// TIA Portal project "Project4" (V17)

(* hardware
DEVICE "S7-1200 station_1"  S7-1200 Station
   slot 0: "Rack_0"  S7-1200 Rack  Rack  V1.0
   slot 1: "PLC_1"  CPU 1212C DC/DC/DC  6ES7 212-1AE40-0XB0  V4.3
DEVICE "HMI_1"  TP1200 Comfort
   slot 0: "HMI_1"  TP1200 Comfort  6AV2 124-0MC01-0AX0  17.0.0.0
   slot 1: "HMI_RT_1"  TP1200 Comfort  6AV2 124-0MC01-0AX0  17.0.0.0
   slot 5: "HMI_1.IE_CP_1"  PROFINET Interface  17.0.0.0
      slot 1: "PROFINET Interface_1"  PROFINET Interface
         slot 1: "Port_1"  Port
         slot 2: "Port_2"  Port
   slot 7: "HMI_1.MPI/DP_CP_1"  MPI/DP Interface  17.0.0.0
*)

// ===== PLC "PLC_1"  CPU 1212C DC/DC/DC =====

VAR_GLOBAL   // PLC tag table "Default tag table"
   "System_Byte" AT %MB1 : Byte;
   "FirstScan" AT %M1.0 : Bool;
   "DiagStatusUpdate" AT %M1.1 : Bool;
   "AlwaysTRUE" AT %M1.2 : Bool;
   "AlwaysFALSE" AT %M1.3 : Bool;
   "Clock_Byte" AT %MB0 : Byte;
   "Clock_10Hz" AT %M0.0 : Bool;
   "Clock_5Hz" AT %M0.1 : Bool;
   "Clock_2.5Hz" AT %M0.2 : Bool;
   "Clock_2Hz" AT %M0.3 : Bool;
   "Clock_1.25Hz" AT %M0.4 : Bool;
   "Clock_1Hz" AT %M0.5 : Bool;
   "Clock_0.625Hz" AT %M0.6 : Bool;
   "Clock_0.5Hz" AT %M0.7 : Bool;
   "Imp1s" AT %M100.0 : Bool;
   "fp_1s" AT %M100.1 : Bool;
   "fp_100ms" AT %M100.2 : Bool;
   "Imp0.1s" AT %M100.3 : Bool;
   "PO1_calc" AT %IW0 : Int;
   "PO2_calc" AT %IW1 : Int;
   "VO1_calc" AT %IW2 : Int;
   "VO2_calc" AT %IW3 : Int;
   "Tag_1" AT %M500.0 : Bool;
   "Tag_2" AT %M500.1 : Bool;
   "Tag_3" AT %M500.2 : Bool;
END_VAR

TYPE "_tSter"
   STRUCT
      Tryb : Bool;
      SterowanieAuto : Bool;
      SterowanieRęka : Bool;
      ZadanaPrędkośćRęka : Int;
      ZadanaPrędkośćAuto : Int;
      PrędkośćWyjściowa : Int;
      Status : Int;
      Wyjscie : Bool;
      CzasWlaczenia : Int;
      Awaria : Bool;
      Ack : Bool;
      "ON/OFF" : Bool;
   END_STRUCT;
END_TYPE

DATA_BLOCK "SterowanieDANE"   // DB1
{ S7_Optimized_Access := 'TRUE' }
VERSION : 0.1
   VAR
      P01 : "_tSter";
      P02 : "_tSter";
      VO1 : "_tSter";
      VO2 : "_tSter";
   END_VAR
BEGIN
   P01.ZadanaPrędkośćAuto := 100;
   P01.PrędkośćWyjściowa := 0;
   P02.ZadanaPrędkośćAuto := 100;
   VO1.ZadanaPrędkośćAuto := 100;
   VO2.ZadanaPrędkośćAuto := 100;
END_DATA_BLOCK

DATA_BLOCK "DB_Zbiornik"   // DB2
{ S7_Optimized_Access := 'TRUE' }
VERSION : 0.1
   VAR
      Poziom : Real;
      LL : Bool;
      LH : Bool;
      PredkoscNapelniania : Int;
      PredkoscOprozniania : Int;
      LM : Bool;
   END_VAR
BEGIN
END_DATA_BLOCK

DATA_BLOCK "Operacje"   // DB4
{ S7_Optimized_Access := 'TRUE' }
VERSION : 0.1
   VAR
      Napelnianie : Bool;
      Oproznianie : Bool;
   END_VAR
BEGIN
END_DATA_BLOCK

DATA_BLOCK "tims"   // DB5
{ S7_Optimized_Access := 'TRUE' }
VERSION : 0.1
   VAR
      ton1 : IEC_TIMER;
      ton2 : IEC_TIMER;
   END_VAR
BEGIN
END_DATA_BLOCK

DATA_BLOCK "Awarie"   // DB6
{ S7_Optimized_Access := 'TRUE' }
VERSION : 0.1
   VAR
      aw : Word;
   END_VAR
BEGIN
END_DATA_BLOCK

// folder: System blocks/Program resources

DATA_BLOCK "IEC_Timer_0_DB"   // DB3
{ S7_Optimized_Access := 'TRUE' }
AUTHOR : Simatic
FAMILY : IEC
NAME : IEC_TMR
VERSION : 1.0
// stored: InstanceOfName IEC_TIMER
"IEC_TIMER"
BEGIN
END_DATA_BLOCK

// folder: (top level)

FUNCTION "FC_Zbiornik" : Void   // FC1, LAD
{ S7_Optimized_Access := 'TRUE' }
VERSION : 0.1
   VAR_IN_OUT
      IEC_Timer_0_Instance : TP_TIME;
   END_VAR
BEGIN

REGION Network 1
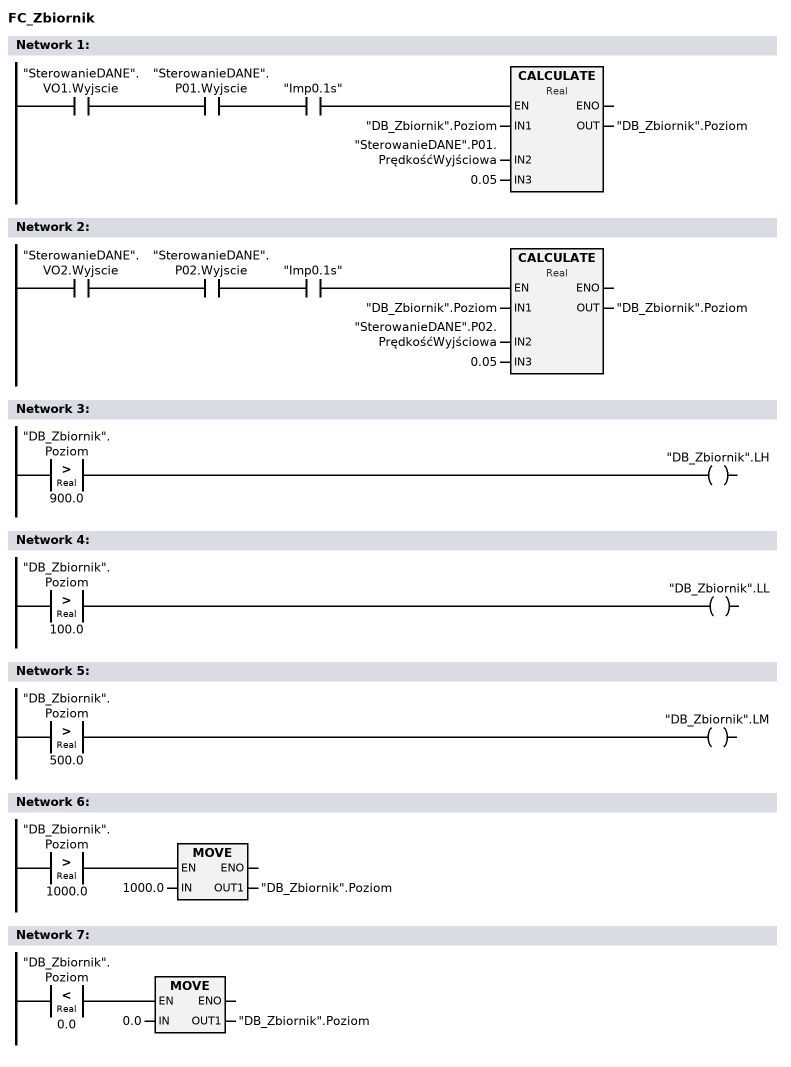
   RUNG wire#powerrail
      Contact( "SterowanieDANE".VO1.Wyjscie )
      Contact( "SterowanieDANE".P01.Wyjscie )
      Contact( "Imp0.1s" )
      { S7_Templates := "SrcType := Real"; S7_Expression := "(IN2 * IN3) + IN1" } Calculate(in1 := "DB_Zbiornik".Poziom, in2 := "SterowanieDANE".P01.PrędkośćWyjściowa, in3 := 0.05, out => "DB_Zbiornik".Poziom)
   END_RUNG
   // the same network as SCL:
   IF "SterowanieDANE".VO1.Wyjscie AND "SterowanieDANE".P01.Wyjscie AND "Imp0.1s" THEN
       "DB_Zbiornik".Poziom := ("SterowanieDANE".P01.PrędkośćWyjściowa * 0.05) + "DB_Zbiornik".Poziom;
   END_IF;
END_REGION

REGION Network 2
   RUNG wire#powerrail
      Contact( "SterowanieDANE".VO2.Wyjscie )
      Contact( "SterowanieDANE".P02.Wyjscie )
      Contact( "Imp0.1s" )
      { S7_Templates := "SrcType := Real"; S7_Expression := "IN1 - (IN2 * IN3)" } Calculate(in1 := "DB_Zbiornik".Poziom, in2 := "SterowanieDANE".P02.PrędkośćWyjściowa, in3 := 0.05, out => "DB_Zbiornik".Poziom)
   END_RUNG
   // the same network as SCL:
   IF "SterowanieDANE".VO2.Wyjscie AND "SterowanieDANE".P02.Wyjscie AND "Imp0.1s" THEN
       "DB_Zbiornik".Poziom := "DB_Zbiornik".Poziom - ("SterowanieDANE".P02.PrędkośćWyjściowa * 0.05);
   END_IF;
END_REGION

REGION Network 3
   RUNG wire#powerrail
      { S7_Templates := "SrcType := Real" } GT_Contact(in1 := "DB_Zbiornik".Poziom, in2 := 900.0)
      Coil( "DB_Zbiornik".LH )
   END_RUNG
   // the same network as SCL:
   "DB_Zbiornik".LH := "DB_Zbiornik".Poziom > 900.0;
END_REGION

REGION Network 4
   RUNG wire#powerrail
      { S7_Templates := "SrcType := Real" } GT_Contact(in1 := "DB_Zbiornik".Poziom, in2 := 100.0)
      Coil( "DB_Zbiornik".LL )
   END_RUNG
   // the same network as SCL:
   "DB_Zbiornik".LL := "DB_Zbiornik".Poziom > 100.0;
END_REGION

REGION Network 5
   RUNG wire#powerrail
      { S7_Templates := "SrcType := Real" } GT_Contact(in1 := "DB_Zbiornik".Poziom, in2 := 500.0)
      Coil( "DB_Zbiornik".LM )
   END_RUNG
   // the same network as SCL:
   "DB_Zbiornik".LM := "DB_Zbiornik".Poziom > 500.0;
END_REGION

REGION Network 6
   RUNG wire#powerrail
      { S7_Templates := "SrcType := Real" } GT_Contact(in1 := "DB_Zbiornik".Poziom, in2 := 1000.0)
      Move(in := 1000.0, out1 => "DB_Zbiornik".Poziom)
   END_RUNG
   // the same network as SCL:
   IF "DB_Zbiornik".Poziom > 1000.0 THEN "DB_Zbiornik".Poziom := 1000.0; END_IF;
END_REGION

REGION Network 7
   RUNG wire#powerrail
      { S7_Templates := "SrcType := Real" } LT_Contact(in1 := "DB_Zbiornik".Poziom, in2 := 0.0)
      Move(in := 0.0, out1 => "DB_Zbiornik".Poziom)
   END_RUNG
   // the same network as SCL:
   IF "DB_Zbiornik".Poziom < 0.0 THEN "DB_Zbiornik".Poziom := 0.0; END_IF;
END_REGION
END_FUNCTION

FUNCTION "Sterowanie" : Void   // FC2, LAD
{ S7_Optimized_Access := 'TRUE' }
VERSION : 0.1
   VAR_INPUT
      ZadanaPrędkośćRęka : Int;
      ZadanaPrędkośćAuto : Int;
      Ack : Bool;
   END_VAR
   VAR_OUTPUT
      PrędkośćWyjściowa : Int;
      Status : Int;
   END_VAR
   VAR_IN_OUT
      "ON/OFF" : Bool;
      Tryb : Bool;
      SterowanieAuto : Bool;
      SterowanieRęka : Bool;
      CzasWlaczenia : Int;
      Awaria : Bool;
      Wyjscie : Bool;
   END_VAR
   VAR_TEMP   // added for the SCL form of the ladder/FBD networks
      _w1 : Bool;
   END_VAR
BEGIN

REGION Network 1: Sterowanie A/R
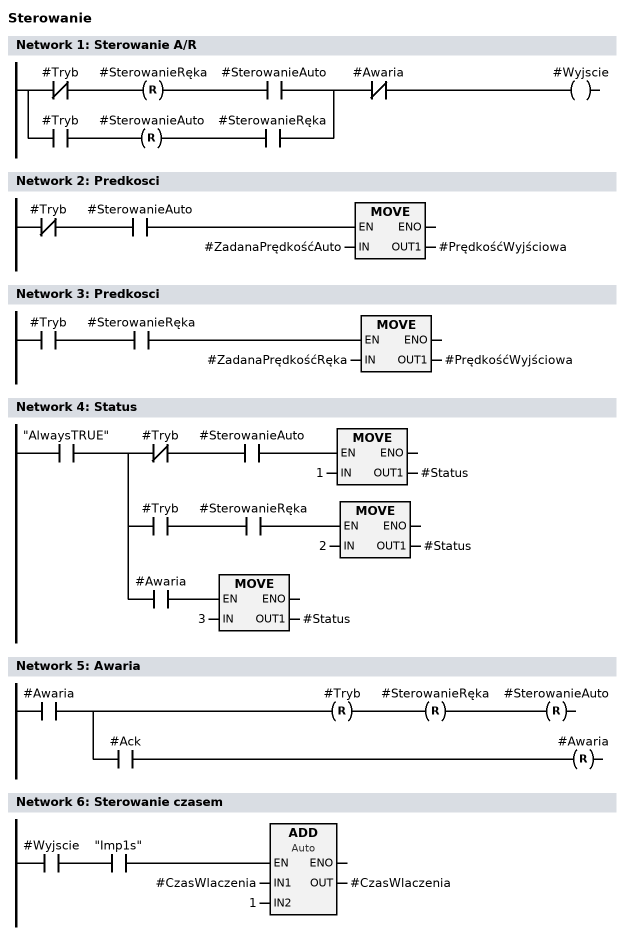
   RUNG wire#powerrail
      I_Contact( #Tryb )
      R_Coil( #SterowanieRęka )
      Contact( #SterowanieAuto )
      wire#w1
      I_Contact( #Awaria )
      Coil( #Wyjscie )
   END_RUNG
   RUNG wire#powerrail
      Contact( #Tryb )
      R_Coil( #SterowanieAuto )
      Contact( #SterowanieRęka )
   END_RUNG wire#w1
   // the same network as SCL:
   IF NOT #Tryb THEN #SterowanieRęka := FALSE; END_IF;
   #_w1 := NOT #Tryb AND #SterowanieAuto;
   IF #Tryb THEN #SterowanieAuto := FALSE; END_IF;
   #Wyjscie := (#_w1 OR (#Tryb AND #SterowanieRęka)) AND NOT #Awaria;
END_REGION

REGION Network 2: Predkosci
   RUNG wire#powerrail
      I_Contact( #Tryb )
      Contact( #SterowanieAuto )
      Move(in := #ZadanaPrędkośćAuto, out1 => #PrędkośćWyjściowa)
   END_RUNG
   // the same network as SCL:
   IF NOT #Tryb AND #SterowanieAuto THEN #PrędkośćWyjściowa := #ZadanaPrędkośćAuto; END_IF;
END_REGION

REGION Network 3: Predkosci
   RUNG wire#powerrail
      Contact( #Tryb )
      Contact( #SterowanieRęka )
      Move(in := #ZadanaPrędkośćRęka, out1 => #PrędkośćWyjściowa)
   END_RUNG
   // the same network as SCL:
   IF #Tryb AND #SterowanieRęka THEN #PrędkośćWyjściowa := #ZadanaPrędkośćRęka; END_IF;
END_REGION

REGION Network 4: Status
   RUNG wire#powerrail
      Contact( "AlwaysTRUE" )
      wire#w1
      I_Contact( #Tryb )
      Contact( #SterowanieAuto )
      Move(in := 1, out1 => #Status)
   END_RUNG
   RUNG wire#w1
      Contact( #Tryb )
      Contact( #SterowanieRęka )
      Move(in := 2, out1 => #Status)
   END_RUNG
   RUNG wire#w1
      Contact( #Awaria )
      Move(in := 3, out1 => #Status)
   END_RUNG
   // the same network as SCL:
   IF "AlwaysTRUE" AND NOT #Tryb AND #SterowanieAuto THEN #Status := 1; END_IF;
   IF "AlwaysTRUE" AND #Tryb AND #SterowanieRęka THEN #Status := 2; END_IF;
   IF "AlwaysTRUE" AND #Awaria THEN #Status := 3; END_IF;
END_REGION

REGION Network 5: Awaria
   RUNG wire#powerrail
      Contact( #Awaria )
      wire#w1
      R_Coil( #Tryb )
      R_Coil( #SterowanieRęka )
      R_Coil( #SterowanieAuto )
   END_RUNG
   RUNG wire#w1
      Contact( #Ack )
      R_Coil( #Awaria )
   END_RUNG
   // the same network as SCL:
   IF #Awaria THEN
       #Tryb := FALSE;
       #SterowanieRęka := FALSE;
       #SterowanieAuto := FALSE;
   END_IF;
   IF #Awaria AND #Ack THEN #Awaria := FALSE; END_IF;
END_REGION

REGION Network 6: Sterowanie czasem
   RUNG wire#powerrail
      Contact( #Wyjscie )
      Contact( "Imp1s" )
      Add(in1 := #CzasWlaczenia, in2 := 1, out => #CzasWlaczenia)
   END_RUNG
   // the same network as SCL:
   IF #Wyjscie AND "Imp1s" THEN #CzasWlaczenia := #CzasWlaczenia + 1; END_IF;
END_REGION
END_FUNCTION

FUNCTION "Napelnianie" : Void   // FC3, LAD
{ S7_Optimized_Access := 'TRUE' }
VERSION : 0.1
BEGIN

REGION Network 1
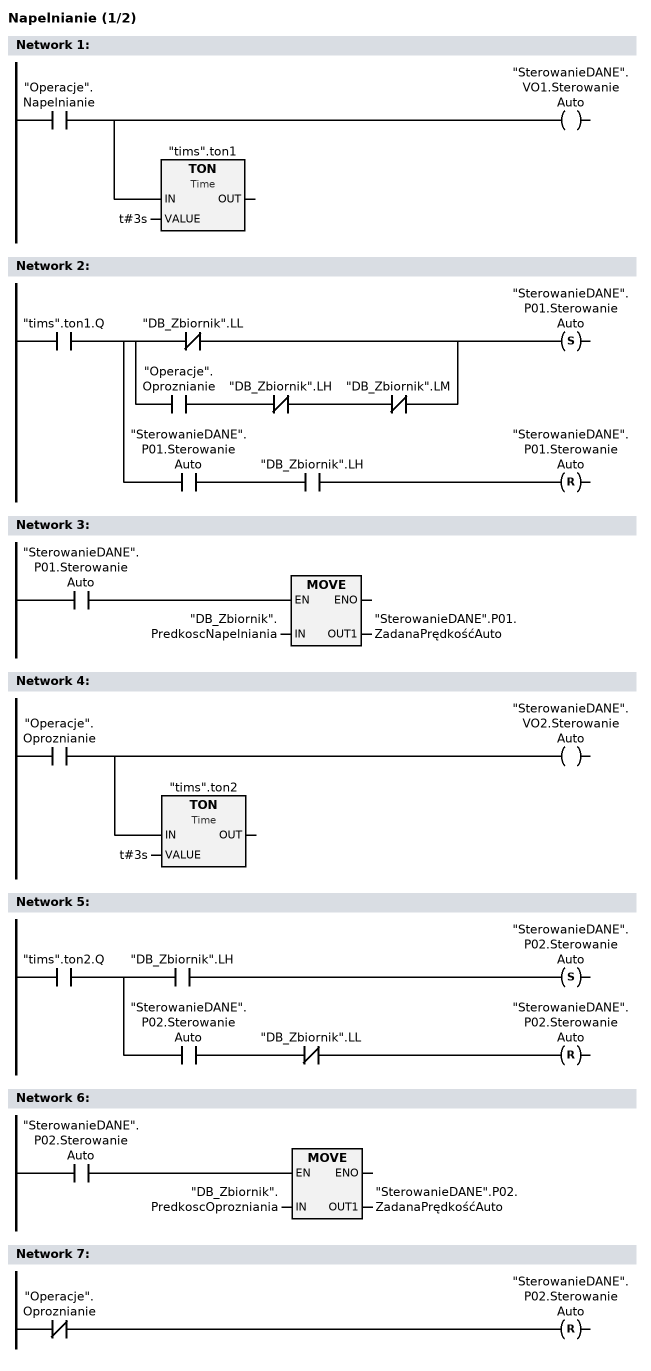
   "SterowanieDANE".VO1.SterowanieAuto := "Operacje".Napelnianie;
   "tims".ton1.TON(IN := "Operacje".Napelnianie, PT := t#3s);   // TON coil
END_REGION

REGION Network 2
   RUNG wire#powerrail
      Contact( "tims".ton1.Q )
      wire#w1
      I_Contact( "DB_Zbiornik".LL )
      wire#w2
      S_Coil( "SterowanieDANE".P01.SterowanieAuto )
   END_RUNG
   RUNG wire#w1
      Contact( "Operacje".Oproznianie )
      I_Contact( "DB_Zbiornik".LH )
      I_Contact( "DB_Zbiornik".LM )
   END_RUNG wire#w2
   RUNG wire#w1
      Contact( "SterowanieDANE".P01.SterowanieAuto )
      Contact( "DB_Zbiornik".LH )
      R_Coil( "SterowanieDANE".P01.SterowanieAuto )
   END_RUNG
   // the same network as SCL:
   IF "tims".ton1.Q AND (NOT "DB_Zbiornik".LL OR ("Operacje".Oproznianie AND NOT "DB_Zbiornik".LH AND NOT "DB_Zbiornik".LM)) THEN
       "SterowanieDANE".P01.SterowanieAuto := TRUE;
   END_IF;
   IF "tims".ton1.Q AND "SterowanieDANE".P01.SterowanieAuto AND "DB_Zbiornik".LH THEN
       "SterowanieDANE".P01.SterowanieAuto := FALSE;
   END_IF;
END_REGION

REGION Network 3
   RUNG wire#powerrail
      Contact( "SterowanieDANE".P01.SterowanieAuto )
      Move(in := "DB_Zbiornik".PredkoscNapelniania, out1 => "SterowanieDANE".P01.ZadanaPrędkośćAuto)
   END_RUNG
   // the same network as SCL:
   IF "SterowanieDANE".P01.SterowanieAuto THEN
       "SterowanieDANE".P01.ZadanaPrędkośćAuto := "DB_Zbiornik".PredkoscNapelniania;
   END_IF;
END_REGION

REGION Network 4
   "SterowanieDANE".VO2.SterowanieAuto := "Operacje".Oproznianie;
   "tims".ton2.TON(IN := "Operacje".Oproznianie, PT := t#3s);   // TON coil
END_REGION

REGION Network 5
   RUNG wire#powerrail
      Contact( "tims".ton2.Q )
      wire#w1
      Contact( "DB_Zbiornik".LH )
      S_Coil( "SterowanieDANE".P02.SterowanieAuto )
   END_RUNG
   RUNG wire#w1
      Contact( "SterowanieDANE".P02.SterowanieAuto )
      I_Contact( "DB_Zbiornik".LL )
      R_Coil( "SterowanieDANE".P02.SterowanieAuto )
   END_RUNG
   // the same network as SCL:
   IF "tims".ton2.Q AND "DB_Zbiornik".LH THEN "SterowanieDANE".P02.SterowanieAuto := TRUE; END_IF;
   IF "tims".ton2.Q AND "SterowanieDANE".P02.SterowanieAuto AND NOT "DB_Zbiornik".LL THEN
       "SterowanieDANE".P02.SterowanieAuto := FALSE;
   END_IF;
END_REGION

REGION Network 6
   RUNG wire#powerrail
      Contact( "SterowanieDANE".P02.SterowanieAuto )
      Move(in := "DB_Zbiornik".PredkoscOprozniania, out1 => "SterowanieDANE".P02.ZadanaPrędkośćAuto)
   END_RUNG
   // the same network as SCL:
   IF "SterowanieDANE".P02.SterowanieAuto THEN
       "SterowanieDANE".P02.ZadanaPrędkośćAuto := "DB_Zbiornik".PredkoscOprozniania;
   END_IF;
END_REGION

REGION Network 7
   RUNG wire#powerrail
      I_Contact( "Operacje".Oproznianie )
      R_Coil( "SterowanieDANE".P02.SterowanieAuto )
   END_RUNG
   // the same network as SCL:
   IF NOT "Operacje".Oproznianie THEN "SterowanieDANE".P02.SterowanieAuto := FALSE; END_IF;
END_REGION

REGION Network 8
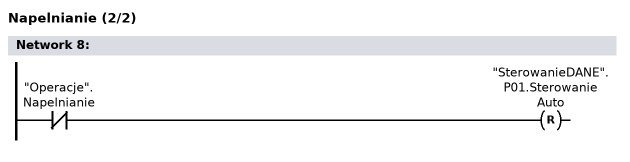
   RUNG wire#powerrail
      I_Contact( "Operacje".Napelnianie )
      R_Coil( "SterowanieDANE".P01.SterowanieAuto )
   END_RUNG
   // the same network as SCL:
   IF NOT "Operacje".Napelnianie THEN "SterowanieDANE".P01.SterowanieAuto := FALSE; END_IF;
END_REGION
END_FUNCTION

ORGANIZATION_BLOCK "Main"   // OB1, LAD, ProgramCycle
TITLE = "Main Program Sweep (Cycle)"
{ S7_Optimized_Access := 'TRUE' }
VERSION : 0.1
   VAR_INPUT
      Initial_Call : Bool;   // Initial call of this OB
      Remanence : Bool;   // =True, if remanent data are available
   END_VAR
   VAR_TEMP   // added for the SCL form of the ladder/FBD networks
      _w1 : Bool;
   END_VAR
BEGIN

REGION Network 1
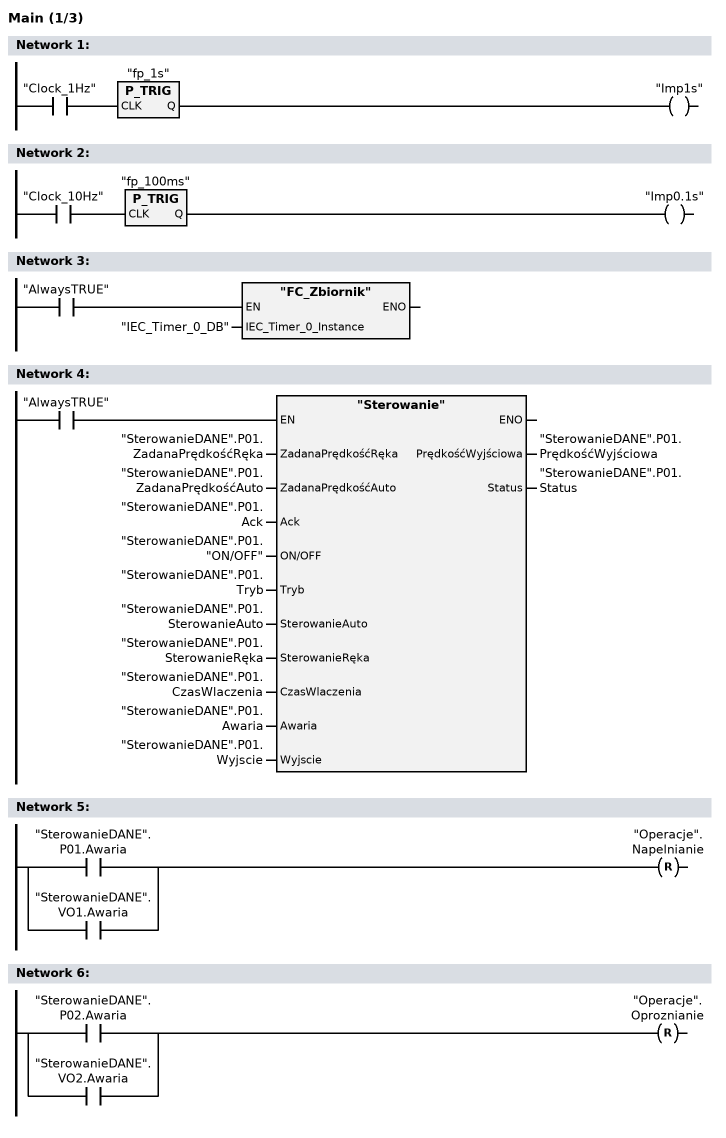
   RUNG wire#powerrail
      Contact( "Clock_1Hz" )
      P_Trig( "fp_1s" )
      Coil( "Imp1s" )
   END_RUNG
   // the same network as SCL:
   #_w1 := "Clock_1Hz" AND NOT "fp_1s";   // rising edge
   "fp_1s" := "Clock_1Hz";
   "Imp1s" := #_w1;
END_REGION

REGION Network 2
   RUNG wire#powerrail
      Contact( "Clock_10Hz" )
      P_Trig( "fp_100ms" )
      Coil( "Imp0.1s" )
   END_RUNG
   // the same network as SCL:
   #_w1 := "Clock_10Hz" AND NOT "fp_100ms";   // rising edge
   "fp_100ms" := "Clock_10Hz";
   "Imp0.1s" := #_w1;
END_REGION

REGION Network 3
   RUNG wire#powerrail
      Contact( "AlwaysTRUE" )
      "FC_Zbiornik"(IEC_Timer_0_Instance := "IEC_Timer_0_DB")
   END_RUNG
   // the same network as SCL:
   IF "AlwaysTRUE" THEN "FC_Zbiornik"(IEC_Timer_0_Instance := "IEC_Timer_0_DB"); END_IF;
END_REGION

REGION Network 4
   RUNG wire#powerrail
      Contact( "AlwaysTRUE" )
      "Sterowanie"(ZadanaPrędkośćRęka := "SterowanieDANE".P01.ZadanaPrędkośćRęka, ZadanaPrędkośćAuto := "SterowanieDANE".P01.ZadanaPrędkośćAuto, Ack := "SterowanieDANE".P01.Ack, "ON/OFF" := "SterowanieDANE".P01."ON/OFF", Tryb := "SterowanieDANE".P01.Tryb, SterowanieAuto := "SterowanieDANE".P01.SterowanieAuto, SterowanieRęka := "SterowanieDANE".P01.SterowanieRęka, CzasWlaczenia := "SterowanieDANE".P01.CzasWlaczenia, Awaria := "SterowanieDANE".P01.Awaria, Wyjscie := "SterowanieDANE".P01.Wyjscie, PrędkośćWyjściowa => "SterowanieDANE".P01.PrędkośćWyjściowa, Status => "SterowanieDANE".P01.Status)
   END_RUNG
   // the same network as SCL:
   IF "AlwaysTRUE" THEN
       "Sterowanie"(ZadanaPrędkośćRęka := "SterowanieDANE".P01.ZadanaPrędkośćRęka,
                    ZadanaPrędkośćAuto := "SterowanieDANE".P01.ZadanaPrędkośćAuto,
                    Ack := "SterowanieDANE".P01.Ack,
                    "ON/OFF" := "SterowanieDANE".P01."ON/OFF",
                    Tryb := "SterowanieDANE".P01.Tryb,
                    SterowanieAuto := "SterowanieDANE".P01.SterowanieAuto,
                    SterowanieRęka := "SterowanieDANE".P01.SterowanieRęka,
                    CzasWlaczenia := "SterowanieDANE".P01.CzasWlaczenia,
                    Awaria := "SterowanieDANE".P01.Awaria,
                    Wyjscie := "SterowanieDANE".P01.Wyjscie,
                    PrędkośćWyjściowa => "SterowanieDANE".P01.PrędkośćWyjściowa,
                    Status => "SterowanieDANE".P01.Status);
   END_IF;
END_REGION

REGION Network 5
   RUNG wire#powerrail
      Contact( "SterowanieDANE".P01.Awaria )
      wire#w1
      R_Coil( "Operacje".Napelnianie )
   END_RUNG
   RUNG wire#powerrail
      Contact( "SterowanieDANE".VO1.Awaria )
   END_RUNG wire#w1
   // the same network as SCL:
   IF "SterowanieDANE".P01.Awaria OR "SterowanieDANE".VO1.Awaria THEN
       "Operacje".Napelnianie := FALSE;
   END_IF;
END_REGION

REGION Network 6
   RUNG wire#powerrail
      Contact( "SterowanieDANE".P02.Awaria )
      wire#w1
      R_Coil( "Operacje".Oproznianie )
   END_RUNG
   RUNG wire#powerrail
      Contact( "SterowanieDANE".VO2.Awaria )
   END_RUNG wire#w1
   // the same network as SCL:
   IF "SterowanieDANE".P02.Awaria OR "SterowanieDANE".VO2.Awaria THEN
       "Operacje".Oproznianie := FALSE;
   END_IF;
END_REGION

REGION Network 7
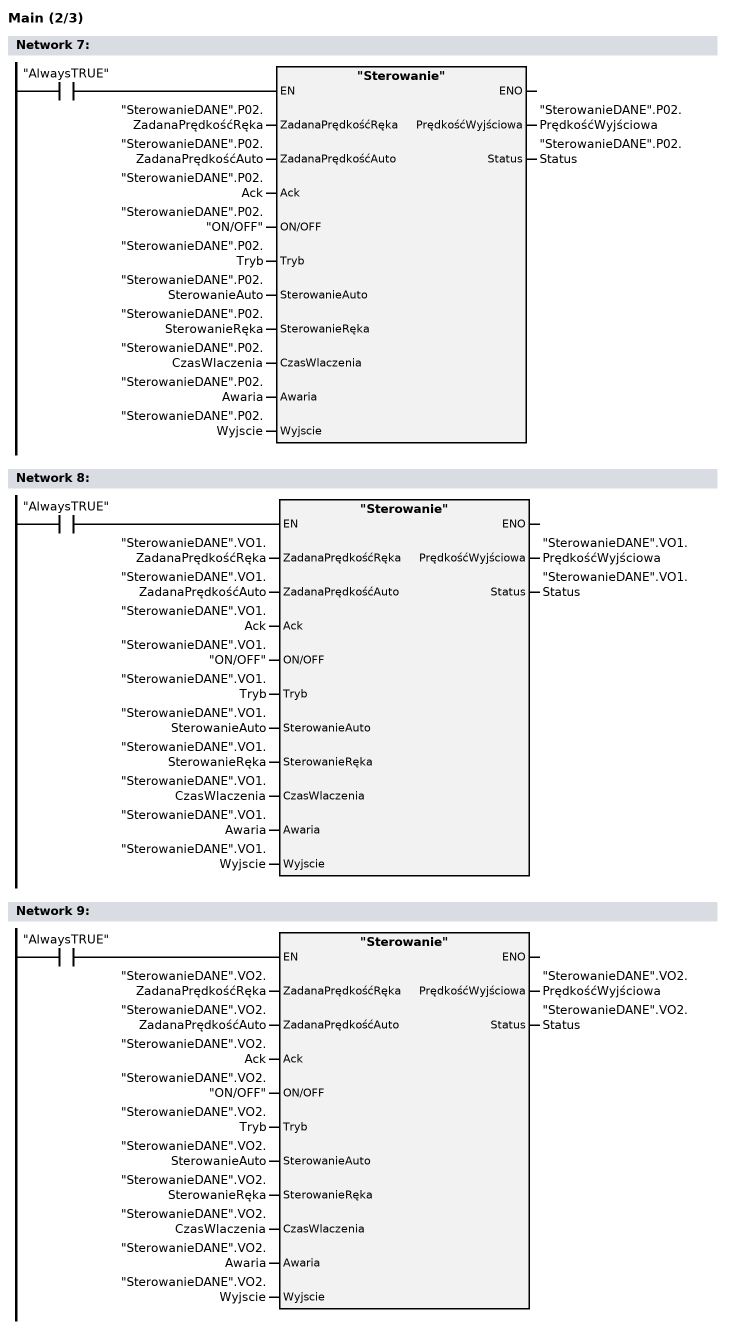
   RUNG wire#powerrail
      Contact( "AlwaysTRUE" )
      "Sterowanie"(ZadanaPrędkośćRęka := "SterowanieDANE".P02.ZadanaPrędkośćRęka, ZadanaPrędkośćAuto := "SterowanieDANE".P02.ZadanaPrędkośćAuto, Ack := "SterowanieDANE".P02.Ack, "ON/OFF" := "SterowanieDANE".P02."ON/OFF", Tryb := "SterowanieDANE".P02.Tryb, SterowanieAuto := "SterowanieDANE".P02.SterowanieAuto, SterowanieRęka := "SterowanieDANE".P02.SterowanieRęka, CzasWlaczenia := "SterowanieDANE".P02.CzasWlaczenia, Awaria := "SterowanieDANE".P02.Awaria, Wyjscie := "SterowanieDANE".P02.Wyjscie, PrędkośćWyjściowa => "SterowanieDANE".P02.PrędkośćWyjściowa, Status => "SterowanieDANE".P02.Status)
   END_RUNG
   // the same network as SCL:
   IF "AlwaysTRUE" THEN
       "Sterowanie"(ZadanaPrędkośćRęka := "SterowanieDANE".P02.ZadanaPrędkośćRęka,
                    ZadanaPrędkośćAuto := "SterowanieDANE".P02.ZadanaPrędkośćAuto,
                    Ack := "SterowanieDANE".P02.Ack,
                    "ON/OFF" := "SterowanieDANE".P02."ON/OFF",
                    Tryb := "SterowanieDANE".P02.Tryb,
                    SterowanieAuto := "SterowanieDANE".P02.SterowanieAuto,
                    SterowanieRęka := "SterowanieDANE".P02.SterowanieRęka,
                    CzasWlaczenia := "SterowanieDANE".P02.CzasWlaczenia,
                    Awaria := "SterowanieDANE".P02.Awaria,
                    Wyjscie := "SterowanieDANE".P02.Wyjscie,
                    PrędkośćWyjściowa => "SterowanieDANE".P02.PrędkośćWyjściowa,
                    Status => "SterowanieDANE".P02.Status);
   END_IF;
END_REGION

REGION Network 8
   RUNG wire#powerrail
      Contact( "AlwaysTRUE" )
      "Sterowanie"(ZadanaPrędkośćRęka := "SterowanieDANE".VO1.ZadanaPrędkośćRęka, ZadanaPrędkośćAuto := "SterowanieDANE".VO1.ZadanaPrędkośćAuto, Ack := "SterowanieDANE".VO1.Ack, "ON/OFF" := "SterowanieDANE".VO1."ON/OFF", Tryb := "SterowanieDANE".VO1.Tryb, SterowanieAuto := "SterowanieDANE".VO1.SterowanieAuto, SterowanieRęka := "SterowanieDANE".VO1.SterowanieRęka, CzasWlaczenia := "SterowanieDANE".VO1.CzasWlaczenia, Awaria := "SterowanieDANE".VO1.Awaria, Wyjscie := "SterowanieDANE".VO1.Wyjscie, PrędkośćWyjściowa => "SterowanieDANE".VO1.PrędkośćWyjściowa, Status => "SterowanieDANE".VO1.Status)
   END_RUNG
   // the same network as SCL:
   IF "AlwaysTRUE" THEN
       "Sterowanie"(ZadanaPrędkośćRęka := "SterowanieDANE".VO1.ZadanaPrędkośćRęka,
                    ZadanaPrędkośćAuto := "SterowanieDANE".VO1.ZadanaPrędkośćAuto,
                    Ack := "SterowanieDANE".VO1.Ack,
                    "ON/OFF" := "SterowanieDANE".VO1."ON/OFF",
                    Tryb := "SterowanieDANE".VO1.Tryb,
                    SterowanieAuto := "SterowanieDANE".VO1.SterowanieAuto,
                    SterowanieRęka := "SterowanieDANE".VO1.SterowanieRęka,
                    CzasWlaczenia := "SterowanieDANE".VO1.CzasWlaczenia,
                    Awaria := "SterowanieDANE".VO1.Awaria,
                    Wyjscie := "SterowanieDANE".VO1.Wyjscie,
                    PrędkośćWyjściowa => "SterowanieDANE".VO1.PrędkośćWyjściowa,
                    Status => "SterowanieDANE".VO1.Status);
   END_IF;
END_REGION

REGION Network 9
   RUNG wire#powerrail
      Contact( "AlwaysTRUE" )
      "Sterowanie"(ZadanaPrędkośćRęka := "SterowanieDANE".VO2.ZadanaPrędkośćRęka, ZadanaPrędkośćAuto := "SterowanieDANE".VO2.ZadanaPrędkośćAuto, Ack := "SterowanieDANE".VO2.Ack, "ON/OFF" := "SterowanieDANE".VO2."ON/OFF", Tryb := "SterowanieDANE".VO2.Tryb, SterowanieAuto := "SterowanieDANE".VO2.SterowanieAuto, SterowanieRęka := "SterowanieDANE".VO2.SterowanieRęka, CzasWlaczenia := "SterowanieDANE".VO2.CzasWlaczenia, Awaria := "SterowanieDANE".VO2.Awaria, Wyjscie := "SterowanieDANE".VO2.Wyjscie, PrędkośćWyjściowa => "SterowanieDANE".VO2.PrędkośćWyjściowa, Status => "SterowanieDANE".VO2.Status)
   END_RUNG
   // the same network as SCL:
   IF "AlwaysTRUE" THEN
       "Sterowanie"(ZadanaPrędkośćRęka := "SterowanieDANE".VO2.ZadanaPrędkośćRęka,
                    ZadanaPrędkośćAuto := "SterowanieDANE".VO2.ZadanaPrędkośćAuto,
                    Ack := "SterowanieDANE".VO2.Ack,
                    "ON/OFF" := "SterowanieDANE".VO2."ON/OFF",
                    Tryb := "SterowanieDANE".VO2.Tryb,
                    SterowanieAuto := "SterowanieDANE".VO2.SterowanieAuto,
                    SterowanieRęka := "SterowanieDANE".VO2.SterowanieRęka,
                    CzasWlaczenia := "SterowanieDANE".VO2.CzasWlaczenia,
                    Awaria := "SterowanieDANE".VO2.Awaria,
                    Wyjscie := "SterowanieDANE".VO2.Wyjscie,
                    PrędkośćWyjściowa => "SterowanieDANE".VO2.PrędkośćWyjściowa,
                    Status => "SterowanieDANE".VO2.Status);
   END_IF;
END_REGION

REGION Network 10
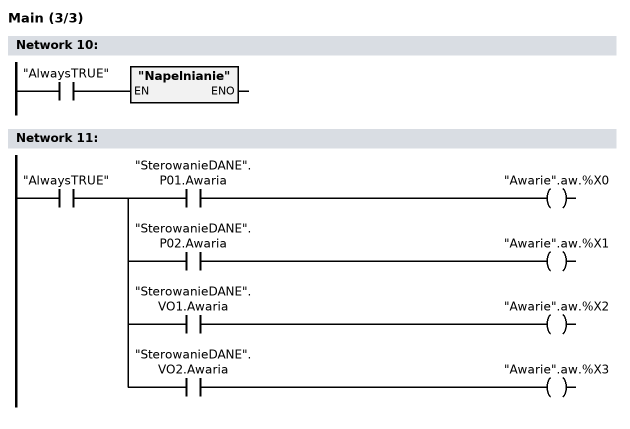
   RUNG wire#powerrail
      Contact( "AlwaysTRUE" )
      "Napelnianie"()
   END_RUNG
   // the same network as SCL:
   IF "AlwaysTRUE" THEN "Napelnianie"(); END_IF;
END_REGION

REGION Network 11
   RUNG wire#powerrail
      Contact( "AlwaysTRUE" )
      wire#w1
      Contact( "SterowanieDANE".P01.Awaria )
      Coil( "Awarie".aw.%X0 )
   END_RUNG
   RUNG wire#w1
      Contact( "SterowanieDANE".P02.Awaria )
      Coil( "Awarie".aw.%X1 )
   END_RUNG
   RUNG wire#w1
      Contact( "SterowanieDANE".VO1.Awaria )
      Coil( "Awarie".aw.%X2 )
   END_RUNG
   RUNG wire#w1
      Contact( "SterowanieDANE".VO2.Awaria )
      Coil( "Awarie".aw.%X3 )
   END_RUNG
   // the same network as SCL:
   "Awarie".aw.%X0 := "AlwaysTRUE" AND "SterowanieDANE".P01.Awaria;
   "Awarie".aw.%X1 := "AlwaysTRUE" AND "SterowanieDANE".P02.Awaria;
   "Awarie".aw.%X2 := "AlwaysTRUE" AND "SterowanieDANE".VO1.Awaria;
   "Awarie".aw.%X3 := "AlwaysTRUE" AND "SterowanieDANE".VO2.Awaria;
END_REGION
END_ORGANIZATION_BLOCK

(* ===== HMI "HMI_RT_1" =====
system functions are stored by id; their names below are inferred from use
connection "HMI_Connection_1": ETHERNET, S7_1200_OMS

HMI tags "Default tag table"
   "SterowaniePompaDANE_PO1_CzasWlaczenia" : Int = PLC SterowanieDANE.P01.CzasWlaczenia AT %DB1.DBW0, 1 s
   "SterowaniePompaDANE_PO1_Tryb" : Bool = PLC SterowanieDANE.P01.Tryb, 1 s
   "SterowaniePompaDANE_PO1_Status" : Int = PLC SterowanieDANE.P01.Status, 1 s
   "SterowaniePompaDANE_PO1_Wyjscie" : Bool = PLC SterowanieDANE.P01.Wyjscie, 1 s
   "SterowaniePompaDANE_PO1_ZadanaPrędkośćRęka" : Int = PLC SterowanieDANE.P01.ZadanaPrędkośćRęka, 1 s
   "SterowaniePompaDANE_PO1_PrędkośćWyjściowa" : Int = PLC SterowanieDANE.P01.PrędkośćWyjściowa, 1 s
   "SterowaniePompaDANE_PO1_SterowanieRęka" : Bool = PLC SterowanieDANE.P01.SterowanieRęka, 1 s
   "PokazCzas" : Bool AT %DB1.DBW0
   "SterowaniePompaDANE_PO1_Awaria" : Bool = PLC SterowanieDANE.P01.Awaria, 1 s
   "SterowanieDANE_P02_Tryb" : Bool = PLC SterowanieDANE.P02.Tryb, 1 s
   "SterowanieDANE_P02_SterowanieRęka" : Bool = PLC SterowanieDANE.P02.SterowanieRęka, 1 s
   "SterowanieDANE_P02_Awaria" : Bool = PLC SterowanieDANE.P02.Awaria, 1 s
   "SterowanieDANE_P02_ZadanaPrędkośćRęka" : Int = PLC SterowanieDANE.P02.ZadanaPrędkośćRęka, 1 s
   "SterowanieDANE_P02_Status" : Int = PLC SterowanieDANE.P02.Status, 1 s
   "PokazCzas2" : Bool AT %DB1.DBW0
   "SterowanieDANE_P02_CzasWlaczenia" : Int = PLC SterowanieDANE.P02.CzasWlaczenia, 1 s
   "SterowanieDANE_P02_PrędkośćWyjściowa" : Int = PLC SterowanieDANE.P02.PrędkośćWyjściowa, 1 s
   "SterowanieDANE_VO1_Tryb" : Bool = PLC SterowanieDANE.VO1.Tryb, 1 s
   "SterowanieDANE_VO1_SterowanieRęka" : Bool = PLC SterowanieDANE.VO1.SterowanieRęka, 1 s
   "SterowanieDANE_VO1_ZadanaPrędkośćRęka" : Int = PLC SterowanieDANE.VO1.ZadanaPrędkośćRęka, 1 s
   "SterowanieDANE_VO1_Awaria" : Bool = PLC SterowanieDANE.VO1.Awaria, 1 s
   "SterowanieDANE_VO1_PrędkośćWyjściowa" : Int = PLC SterowanieDANE.VO1.PrędkośćWyjściowa, 1 s
   "SterowanieDANE_VO1_CzasWlaczenia" : Int = PLC SterowanieDANE.VO1.CzasWlaczenia, 1 s
   "PokazCzas3" : Bool AT %DB1.DBW0
   "PokazCzas4" : Bool AT %DB1.DBW0
   "SterowanieDANE_VO2_Tryb" : Bool = PLC SterowanieDANE.VO2.Tryb, 1 s
   "SterowanieDANE_VO2_ZadanaPrędkośćRęka" : Int = PLC SterowanieDANE.VO2.ZadanaPrędkośćRęka, 1 s
   "SterowanieDANE_VO2_PrędkośćWyjściowa" : Int = PLC SterowanieDANE.VO2.PrędkośćWyjściowa, 1 s
   "SterowanieDANE_VO2_Status" : Int = PLC SterowanieDANE.VO2.Status, 1 s
   "SterowanieDANE_VO2_CzasWlaczenia" : Int = PLC SterowanieDANE.VO2.CzasWlaczenia, 1 s
   "SterowanieDANE_VO2_Awaria" : Bool = PLC SterowanieDANE.VO2.Awaria, 1 s
   "SterowanieDANE_VO1_Status" : Int = PLC SterowanieDANE.VO1.Status, 1 s
   "SterowanieDANE_VO2_SterowanieRęka" : Bool = PLC SterowanieDANE.VO2.SterowanieRęka, 1 s
   "SterowanieDANE_P01_ON/OFF" : Bool = PLC SterowanieDANE.P01.ON/OFF, 1 s
   "SterowanieDANE_P02_ON/OFF" : Bool = PLC SterowanieDANE.P02.ON/OFF, 1 s
   "SterowanieDANE_VO1_ON/OFF" : Bool = PLC SterowanieDANE.VO1.ON/OFF, 1 s
   "SterowanieDANE_VO2_ON/OFF" : Bool = PLC SterowanieDANE.VO2.ON/OFF, 1 s
   "DB_Zbiornik_Poziom" : Real = PLC DB_Zbiornik.Poziom, 100 ms
   "SterowanieDANE_P02_Wyjscie" : Bool = PLC SterowanieDANE.P02.Wyjscie, 1 s
   "SterowanieDANE_VO1_Wyjscie" : Bool = PLC SterowanieDANE.VO1.Wyjscie, 1 s
   "SterowanieDANE_VO2_Wyjscie" : Bool = PLC SterowanieDANE.VO2.Wyjscie, 1 s
   "DB_Zbiornik_LH" : Bool = PLC DB_Zbiornik.LH, 1 s
   "DB_Zbiornik_LL" : Bool = PLC DB_Zbiornik.LL, 1 s
   "Operacje_Napelnianie" : Bool = PLC Operacje.Napelnianie, 1 s
   "Operacje_Oproznianie" : Bool = PLC Operacje.Oproznianie, 1 s
   "DB_Zbiornik_PredkoscNapelniania" : Int = PLC DB_Zbiornik.PredkoscNapelniania, 1 s
   "DB_Zbiornik_PredkoscOprozniania" : Int = PLC DB_Zbiornik.PredkoscOprozniania, 1 s
   "DB_Zbiornik_LM" : Bool = PLC DB_Zbiornik.LM, 1 s
   "Awarie_aw" : Word = PLC Awarie.aw, 1 s
   "SterowanieDANE_VO2_Ack" : Bool = PLC SterowanieDANE.VO2.Ack, 1 s
   "SterowanieDANE_VO1_Ack" : Bool = PLC SterowanieDANE.VO1.Ack, 1 s
   "SterowanieDANE_P01_Ack" : Bool = PLC SterowanieDANE.P01.Ack, 1 s

discrete alarms
   1: 'Awaria pompy P01', class Errors, trigger "Awarie_aw" bit 0
   2: 'Awaria pompy P02', class Errors, trigger "Awarie_aw" bit 1
   3: 'Awaria zaworu v01', class Errors, trigger "Awarie_aw" bit 2
   4: 'Awaria zaworu v02', class Errors, trigger "Awarie_aw" bit 3

graphic list "Pompa": 0 'Graphic_3'; 1 'Graphic_1'; 2 'Graphic_4'; 3 'Graphic_5'

graphic list "Zawory": 0 'Graphic_11'; 1 'Graphic_10'; 2 'Graphic_12'; 3 'Graphic_13'

graphic list "ZaworySciezka": 0 'Graphic_20'; 1 'Graphic_18'

graphic list "PoziomWody": 0 'Graphic_21'

screen "SterowanieReczne" 1280x799, template "Template_1"
   on GenerateScreen: SetTag("SterowaniePompaDANE_PO1_CzasWlaczenia", 1)
   Switch "Switch_1" at 28,120 size 75x75; CaptionText 'Auto/Ręka'; TextOff 'Auto'; TextOn 'Ręka'
      ProcessValue <- "SterowaniePompaDANE_PO1_Tryb"
   GraphicIOField "Graphic I/O field_1" at 282,138 size 65x61; PictureList "Pompa"
      ProcessValue <- "SterowaniePompaDANE_PO1_Status"
   IOField "I/O field_1" at 258,209 size 96x32; FormatPattern s99999
      ProcessValue <- "SterowaniePompaDANE_PO1_PrędkośćWyjściowa"
   IOField "I/O field_2" at 168,141 size 89x51; FormatPattern s99999
      Visibility <- "SterowaniePompaDANE_PO1_Tryb"
      ProcessValue <- "SterowaniePompaDANE_PO1_ZadanaPrędkośćRęka"
   Switch "Switch_3" at 105,141 size 53x53; CaptionText 'Switch'; TextOff 'OFF'; TextOn 'ON'
      ProcessValue <- "SterowaniePompaDANE_PO1_SterowanieRęka"
      Visibility <- "SterowaniePompaDANE_PO1_Tryb"
   Rectangle "Rectangle_1" at 396,141 size 143x119
      Visibility <- "PokazCzas"
   TextField "Text field_1" at 397,147 size 154x25; Text 'Czas Zalaczenia'
      Visibility <- "PokazCzas"
   IOField "I/O field_3" at 419,172 size 96x34; FormatPattern s99999
      ProcessValue <- "SterowaniePompaDANE_PO1_CzasWlaczenia"
      Visibility <- "PokazCzas"
   TextField "Text field_2" at 517,176 size 15x25; Text 's'
      Visibility <- "PokazCzas"
   TextField "Text field_3" at 358,213 size 26x25; Text '%'
   TextField "Text field_4" at 258,154 size 26x25; Text '%'
      Visibility <- "SterowaniePompaDANE_PO1_Tryb"
   Switch "Switch_2" at 352,166 size 38x36; CaptionText 'Switch'; TextOff 'OFF'; TextOn 'ON'; PictureOn "Graphic_6"; PictureOff "Graphic_6"
      ProcessValue <- "PokazCzas"
   Button "Button_1" at 439,211 size 58x36; TextOff 'reset'
      on Press: SetTag("SterowaniePompaDANE_PO1_CzasWlaczenia", 0)
      Visibility <- "PokazCzas"
   Button "Button_3" at 28,209 size 73x51; TextOff 'Awaria'
      on Change: SetTag("SterowaniePompaDANE_PO1_Awaria", 1)
      Appearance <- "SterowaniePompaDANE_PO1_Awaria"
   Button "Button_4" at 105,211 size 132x50; TextOff 'Wylacz awarie'
      on Change: SetTag("SterowanieDANE_P01_Ack", 1)
      Visibility <- "SterowaniePompaDANE_PO1_Awaria"
   Switch "Switch_4" at 28,295 size 75x75; TextOn 'Ręka'; CaptionText 'Auto/Ręka'; TextOff 'Auto'
      ProcessValue <- "SterowanieDANE_P02_Tryb"
   IOField "I/O field_4" at 253,385 size 96x32; FormatPattern s99999
      ProcessValue <- "SterowanieDANE_P02_PrędkośćWyjściowa"
   IOField "I/O field_5" at 161,318 size 87x51; FormatPattern s99999
      ProcessValue <- "SterowanieDANE_P02_ZadanaPrędkośćRęka"
      Visibility <- "SterowanieDANE_P02_Tryb"
   GraphicIOField "Graphic I/O field_2" at 279,314 size 65x61; PictureList "Pompa"
      ProcessValue <- "SterowanieDANE_P02_Status"
   Switch "Switch_5" at 105,316 size 51x53; TextOn 'ON'; CaptionText 'Switch'; TextOff 'OFF'
      ProcessValue <- "SterowanieDANE_P02_SterowanieRęka"
      Visibility <- "SterowanieDANE_P02_Tryb"
   Rectangle "Rectangle_4" at 396,305 size 146x119
      Visibility <- "PokazCzas2"
   TextField "Text field_6" at 396,305 size 154x25; Text 'Czas Zalaczenia'
      Visibility <- "PokazCzas2"
   IOField "I/O field_6" at 423,331 size 96x34; FormatPattern s99999
      Visibility <- "PokazCzas2"
      ProcessValue <- "SterowanieDANE_P02_CzasWlaczenia"
   TextField "Text field_7" at 524,336 size 15x25; Text 's'
      Visibility <- "PokazCzas2"
   TextField "Text field_8" at 250,330 size 26x25; Text '%'
   TextField "Text field_9" at 352,389 size 26x25; Text '%'
      Visibility <- "SterowaniePompaDANE_PO1_Tryb"
   Switch "Switch_6" at 349,343 size 38x36; CaptionText 'Switch'; TextOff 'OFF'; TextOn 'ON'; PictureOff "Graphic_6"; PictureOn "Graphic_6"
      ProcessValue <- "PokazCzas2"
   Button "Button_5" at 438,370 size 58x36; TextOff 'reset'
      on Press: SetTag("SterowanieDANE_P02_CzasWlaczenia", 0)
      Visibility <- "PokazCzas2"
   Button "Button_6" at 26,379 size 75x51; TextOff 'Awaria'
      on Change: SetTag("SterowanieDANE_P02_Awaria", 1)
      Appearance <- "SterowanieDANE_P02_Awaria"
   Button "Button_7" at 106,379 size 127x50; TextOff 'Wylacz awarie'
      on Change: SetTag("SterowanieDANE_VO1_Ack", 1)
      Visibility <- "SterowanieDANE_P02_Awaria"
   Switch "Switch_7" at 28,460 size 74x75; TextOn 'Ręka'; CaptionText 'Auto/Ręka'; TextOff 'Auto'
      ProcessValue <- "SterowanieDANE_VO1_Tryb"
   GraphicIOField "Graphic I/O field_3" at 282,479 size 65x61; PictureList "Zawory"
      ProcessValue <- "SterowanieDANE_VO1_Status"
   Switch "Switch_8" at 105,480 size 54x53; TextOn 'ON'; CaptionText 'Switch'; TextOff 'OFF'
      ProcessValue <- "SterowanieDANE_VO1_SterowanieRęka"
      Visibility <- "SterowanieDANE_VO1_Tryb"
   Rectangle "Rectangle_7" at 397,463 size 147x119
      Visibility <- "PokazCzas3"
   TextField "Text field_12" at 404,466 size 154x25; Text 'Czas Zalaczenia'
      Visibility <- "PokazCzas3"
   IOField "I/O field_9" at 424,498 size 96x34; FormatPattern s99999
      ProcessValue <- "SterowanieDANE_VO1_CzasWlaczenia"
      Visibility <- "PokazCzas3"
   TextField "Text field_13" at 526,498 size 15x25; Text 's'
      Visibility <- "PokazCzas3"
   Switch "Switch_9" at 352,501 size 38x36; CaptionText 'Switch'; TextOff 'OFF'; TextOn 'ON'; PictureOff "Graphic_6"; PictureOn "Graphic_6"
      ProcessValue <- "PokazCzas3"
   Button "Button_8" at 443,537 size 58x36; TextOff 'reset'
      on Press: SetTag("SterowanieDANE_VO1_CzasWlaczenia", 0)
      Visibility <- "PokazCzas3"
   Button "Button_9" at 28,549 size 104x51; TextOff 'Awaria'
      on Change: SetTag("SterowanieDANE_VO1_Awaria", 1)
      Appearance <- "SterowanieDANE_VO1_Awaria"
   Button "Button_10" at 135,549 size 112x50; TextOff 'Wylacz awarie'
      on Change: SetTag("SterowanieDANE_VO1_Ack", 1)
      Visibility <- "SterowanieDANE_VO1_Awaria"
   Switch "Switch_10" at 26,637 size 84x75; TextOn 'Ręka'; CaptionText 'Auto/Ręka'; TextOff 'Auto'
      ProcessValue <- "SterowanieDANE_VO2_Tryb"
   GraphicIOField "Graphic I/O field_4" at 284,653 size 65x61; PictureList "Zawory"
      ProcessValue <- "SterowanieDANE_VO2_Status"
   Switch "Switch_11" at 113,659 size 53x53; TextOn 'ON'; CaptionText 'Switch'; TextOff 'OFF'
      ProcessValue <- "SterowanieDANE_VO2_SterowanieRęka"
      Visibility <- "SterowanieDANE_VO2_Tryb"
   Rectangle "Rectangle_8" at 399,637 size 143x119
      Visibility <- "PokazCzas4"
   TextField "Text field_16" at 405,642 size 154x25; Text 'Czas Zalaczenia'
      Visibility <- "PokazCzas4"
   IOField "I/O field_12" at 428,675 size 96x34; FormatPattern s99999
      ProcessValue <- "SterowanieDANE_VO2_CzasWlaczenia"
      Visibility <- "PokazCzas4"
   TextField "Text field_18" at 528,678 size 15x25; Text 's'
      Visibility <- "PokazCzas4"
   Switch "Switch_12" at 353,678 size 38x36; CaptionText 'Switch'; TextOff 'OFF'; TextOn 'ON'; PictureOff "Graphic_6"; PictureOn "Graphic_6"
      ProcessValue <- "PokazCzas4"
   Button "Button_11" at 442,712 size 58x36; TextOff 'reset'
      on Press: SetTag("SterowanieDANE_VO2_CzasWlaczenia", 0)
      Visibility <- "PokazCzas4"
   Button "Button_12" at 26,726 size 104x51; TextOff 'Awaria'
      on Change: SetTag("SterowanieDANE_VO2_Awaria", 1)
      Appearance <- "SterowanieDANE_VO2_Awaria"
   Button "Button_13" at 134,726 size 118x50; TextOff 'Wylacz awarie'
      on Change: SetTag("SterowanieDANE_VO2_Ack", 1)
      Visibility <- "SterowanieDANE_VO2_Awaria"
   TextField "Text field_17" at 298,109 size 41x25; Text 'P01'
   TextField "Text field_5" at 300,284 size 41x25; Text 'P02'
   TextField "Text field_10" at 297,455 size 41x25; Text 'V01'
   TextField "Text field_11" at 300,630 size 41x25; Text 'V02'
   Line "Line_1" at 647,544 size 48x0
      Appearance <- "SterowaniePompaDANE_PO1_Wyjscie"
   Line "Line_2" at 724,467 size 0x42
      Appearance <- "SterowanieDANE_VO1_Wyjscie"
   Line "Line_4" at 758,541 size 44x0
      Appearance <- "SterowanieDANE_VO1_Wyjscie"
   GraphicIOField "Graphic I/O field_5" at 581,514 size 65x58; PictureList "Pompa"
      ProcessValue <- "SterowaniePompaDANE_PO1_Status"
   GraphicIOField "Graphic I/O field_6" at 690,400 size 78x65; PictureList "Zawory"
      ProcessValue <- "SterowanieDANE_VO1_Status"
   TextField "Text field_21" at 591,490 size 43x25; Text 'PO1'
   TextField "Text field_22" at 709,372 size 43x25; Text 'VO1'
   GraphicIOField "Graphic I/O field_7" at 691,508 size 68x64; PictureList "ZaworySciezka"
      ProcessValue <- "SterowanieDANE_VO1_Wyjscie"
   Line "Line_8" at 978,545 size 76x0
      Appearance <- "SterowanieDANE_VO2_Wyjscie"
   Line "Line_9" at 1076,456 size 0x52
      Appearance <- "SterowanieDANE_VO2_Wyjscie"
   Bar "Bar_1" at 801,199 size 190x376; MinimumValue 0; MaximumValue 1000
      ProcessValue <- "DB_Zbiornik_Poziom"
   Line "Line_11" at 1096,544 size 74x0
      Appearance <- "SterowanieDANE_P02_Wyjscie"
   GraphicIOField "Graphic I/O field_8" at 1166,512 size 72x63; PictureList "Pompa"
      ProcessValue <- "SterowanieDANE_P02_Status"
   GraphicIOField "Graphic I/O field_9" at 1037,397 size 78x68; PictureList "Zawory"
      ProcessValue <- "SterowanieDANE_VO2_Status"
   TextField "Text field_23" at 1179,486 size 43x25; Text 'PO2'
   TextField "Text field_24" at 1054,370 size 43x25; Text 'VO2'
   GraphicIOField "Graphic I/O field_10" at 1040,512 size 69x63; PictureList "ZaworySciezka"
      ProcessValue <- "SterowanieDANE_VO2_Wyjscie"
   Line "Line_3" at 946,244 size 40x0
      Appearance <- "DB_Zbiornik_LH"
   Circle "Circle_1" at 978,227 size 33x33
      Appearance <- "DB_Zbiornik_LH"
   Line "Line_5" at 920,545 size 40x0
      Appearance <- "DB_Zbiornik_LL"
   Circle "Circle_2" at 958,523 size 39x39
      Appearance <- "DB_Zbiornik_LL"
   Switch "Switch_13" at 604,104 size 120x88; CaptionText 'Napelnianie'; TextOff 'OFF'; TextOn 'ON'
      ProcessValue <- "Operacje_Napelnianie"
   Switch "Switch_14" at 1065,100 size 120x88; CaptionText 'Oproznianie'; TextOff 'OFF'; TextOn 'ON'
      ProcessValue <- "Operacje_Oproznianie"
   Slider "Slider_1" at 589,195 size 80x230; Caption 'SIMATIC'
      ProcessValue <- "DB_Zbiornik_PredkoscNapelniania"
   Slider "Slider_2" at 1142,188 size 80x230; Caption 'SIMATIC'
      ProcessValue <- "DB_Zbiornik_PredkoscOprozniania"
   Line "Line_6" at 942,390 size 40x0
      Appearance <- "DB_Zbiornik_LH"
   Circle "Circle_3" at 974,373 size 33x33
      Appearance <- "DB_Zbiornik_LM"

Template "Template_1" 1280x799
   AlarmView "Template_Alarm view_1" at 0,1 size 1277x100
*)